# EPICS substitutions: template/sensor_cpu_ess.substitutions
#
# NAT MCH Sensor PV
# nat> show_sensorinfo 5
# Sensor Information for FRU 5 / AMC1
# ==================================================================
#   #   SDRType  Sensor Entity Inst  Value   State    Name
# ------------------------------------------------------------------
#   -   MDevLoc          0xc1  0x61                    CCT AM 900/412
#     - unknown SDR=0x13
#     - unknown SDR=0x13  2   Full     Temp    0xc1  0x61  39 C       ok     CPU INT Temp
#   3   Full     Temp    0xc1  0x61  40 C       ok     CPU AMB Temp
#   4   Full     Temp    0xc1  0x61  39 C       ok     Ambient Temp
#   5   Full     Voltage 0xc1  0x61  12.354 V   ok     +12V PSU
#   6   Full     Voltage 0xc1  0x61  5.146 V    ok     +5V PSU
#   7   Full     Voltage 0xc1  0x61  3.249 V    ok     +3.3V PSU
#   8   Full     Voltage 0xc1  0x61  1.090 V    ok     +PS 1V05
#   9   Full     Voltage 0xc1  0x61  1.010 V    ok     +PS 1V0
#  10   Full     Voltage 0xc1  0x61  0.660 V    ok     VCC CORE
#  11   Compact  0xf2    0xc1  0x61  0x01              Ejector Handle
#  12   Compact  0xf0    0xc1  0x61  0x10              HS 005 AMC1
# ------------------------------------------------------------------

global {dev=$(dev), id=CPU, unit=$(unit), fruid=$(fruid), prefix=$(id)$(unit)}

file "sensor_ai_ess.template"
{
   pattern { attr	, sensinst	, type	}
           { TEMP	, 1		, 1	}
           { TEMP	, 2		, 1	}
           { V		, 1		, 2	}
           { V		, 2		, 2	}
           { V		, 3		, 2	}
           { V		, 4		, 2	}
           { V		, 5		, 2	}
           { V		, 6		, 2	}
}
